FUNCTION TryConvert_LINT_TO_UDINT : BOOL
VAR_INPUT
	in : LINT;
	out : REFERENCE TO UDINT;
END_VAR

IF in > DatatypeLimits.MAX_VALUE_OF_LINT_WHICH_CAN_BE_HELD_IN_A_UDINT THEN
	RETURN;
END_IF

IF in < DatatypeLimits.MIN_VALUE_OF_LINT_WHICH_CAN_BE_HELD_IN_A_UDINT THEN
	RETURN;
END_IF

out := LINT_TO_UDINT(in);
TryConvert_LINT_TO_UDINT := TRUE;

END_FUNCTION

(* stored: Version 1.1.0.1, ProductVersion 3.1.4024.12
   POU TryConvert_LINT_TO_UDINT: Id {c6ca1782-0da6-4599-9aa4-a0a28348d251}, SpecialFunc None *)
